FUNCTION_BLOCK AD_TO_AUDI (* Composite FB for converting AD (DWORD) adapter to AUDI (UDINT) adapter *)
  (* Standard: 61499-2; Description: Copyright (c) 2026 HR Agrartechnik GmbH This program and the accompanying materials are made available under the terms of the Eclipse Public License 2.0 which is available at https://www.eclipse.org/legal/epl-2.0/ SPDX-License-Identifier: EPL-2.0 *)
  (* Version 1.0, 2026-01-17, Franz Hoepfinger, HR Agrartechnik GmbH *)
  PACKAGE adapter::conversion::unidirectional;
  IMPORT eclipse4diac::core::TypeHash;
  IMPORT iec61131::conversion::F_DWORD_TO_UDINT;
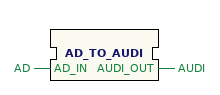
  SOCKETS
    AD_IN : adapter::types::unidirectional::AD; (* DWORD Adapter Input *)
  END_SOCKETS
  PLUGS
    AUDI_OUT : adapter::types::unidirectional::AUDI; (* UDINT Adapter Output *)
  END_PLUGS
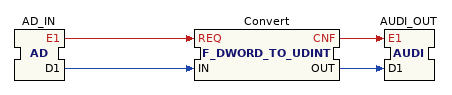
  FBS
    Convert : iec61131::conversion::F_DWORD_TO_UDINT;
  END_FBS
  EVENT_CONNECTIONS
    AD_IN.E1 TO Convert.REQ;
    Convert.CNF TO AUDI_OUT.E1;
  END_CONNECTIONS
  DATA_CONNECTIONS
    AD_IN.D1 TO Convert.IN;
    Convert.OUT TO AUDI_OUT.D1;
  END_CONNECTIONS
END_FUNCTION_BLOCK
